TYPE
    TcoInsightConfig_v_5_x_x :
    STRUCT
        ResultDataSize : eTcoInsightResultDataSize_v_5_x_x := eTcoInsightResultDataSize_v_5_x_x.RESULT_DATA_64B;
        UserDataSize : eTcoInsightUserDataSize_v_5_x_x := eTcoInsightUserDataSize_v_5_x_x.USER_DATA_64B;
        DataFormat : eTcoDataFormat := TcoUtilities.eTcoDataFormat.BigEndian;
        MaxJobNumber : UINT := 999;
        InfoTime : TIME := T#2S;
        ErrorTime : TIME := T#5S;
    //	ServiceJobNumber		:	UINT;
    //	ServiceJobName			:	STRING;
    //	ServiceSoftEventNumber	:	UINT;
    END_STRUCT
END_TYPE

(* stored: Version 1.1.0.1, ProductVersion 3.1.4024.10
   DUT TcoInsightConfig_v_5_x_x: Id {4f2c0f1b-fa0b-09ae-14c5-7f6db18badfb} *)
